(* IEC 61131-3 sources: 89152_FlorisHendrix_AfstudeerProject/89152_FlorisHendrix_ExamenProject/Stations/MachineControl/MachineControl/Class/_QuitErrorLMCaxis, 1 file *)

(* ---- _QuitErrorLMCaxis.st ---- *)
(*!
<Class
	Name               = "_QuitErrorLMCaxis"
	Revision           = "1.0"
	RealtimeTask       = "false"
	CyclicTask         = "false"
	BackgroundTask     = "false"
	Sigmatek           = "true"
	OSInterface        = "false"
	HighPriority       = "false"
	Automatic          = "false"
	UpdateMode         = "Prescan"
	SharedCommandTable = "true"
	Objectsize         = "(374,120)">
	<Channels>
		<Server Name="ClassSvr" Visualized="false" Initialize="false" WriteProtected="false" Retentive="false"/>
		<Client Name="LMCAXIS" Required="false" Internal="false"/>
	</Channels>
	<Dependencies>
		<Files>
			<File Path=".\Class\_QuitErrorLMCaxis\_QuitErrorLMCAxis_de.pdf"/>
			<File Path=".\Class\_QuitErrorLMCaxis\_QuitErrorLMCAxis_en.pdf"/>
		</Files>
	</Dependencies>
	<RevDoku>
		<Owner Company="Sigmatek" Author="roskri"/>
		<Dokumentation Revision="1.0" Date="2016-07-07" Author="roskri" Company="Sigmatek" Description="Class added for quitting error on _LMCAxis"/>
	</RevDoku>
</Class>
*)
_QuitErrorLMCaxis : CLASS
  //Servers:
	ClassSvr 	: SvrChCmd_DINT;
  //Clients:
	LMCAXIS 	: CltChCmd__LMCAxis;
  //Variables:
		bClientConnected 	: BOOL;
  //Functions:

	FUNCTION VIRTUAL GLOBAL Init;

	FUNCTION VIRTUAL GLOBAL ClassSvr::Write
		VAR_INPUT
			input (EAX) 	: DINT;
		END_VAR
		VAR_OUTPUT
			result (EAX) 	: DINT;
		END_VAR;
  //Tables:
	FUNCTION @STD
		VAR_OUTPUT
			ret_code	: CONFSTATES;
		END_VAR;
	FUNCTION GLOBAL TAB @CT_;
END_CLASS;

#pragma usingLtd _LMCAxis

FUNCTION VIRTUAL GLOBAL _QuitErrorLMCAxis::ClassSvr::Write
	VAR_INPUT
		input (EAX) 	: DINT;
	END_VAR
	VAR_OUTPUT
		result (EAX) 	: DINT;
	END_VAR

	ClassSvr := input;
	result := ClassSvr;

  if ClassSvr = 1 & bClientConnected then
    LMCAXIS.QuitError();
  end_if;

END_FUNCTION

FUNCTION VIRTUAL GLOBAL _QuitErrorLMCAxis::Init

  if _FirstScan then
    if IsClientConnected(#LMCAXIS) then
      bClientConnected := TRUE;
    end_if;
  end_if;

END_FUNCTION
